TYPE (* logiBUS DO Struct Octal *)
  (* Version 1.0, 2026-05-28, franz *)
  PACKAGE logiBUS::io::DQ;
  IMPORT logiBUS::io::DQ::logiBUS_DO_S;
  logiBUS_DO_S_Octal : STRUCT
    Port1 : logiBUS_DO_S := (Pin := 255);
    Port2 : logiBUS_DO_S := (Pin := 255);
    Port3 : logiBUS_DO_S := (Pin := 255);
    Port4 : logiBUS_DO_S := (Pin := 255);
    Port5 : logiBUS_DO_S := (Pin := 255);
    Port6 : logiBUS_DO_S := (Pin := 255);
    Port7 : logiBUS_DO_S := (Pin := 255);
    Port8 : logiBUS_DO_S := (Pin := 255);
  END_STRUCT;
END_TYPE
